KUKA KRL program: end_weld_respot.src

&ACCESS RVO3
&REL 155
&COMMENT end_weld_RESPOT
&PARAM DISKPATH = KRC:\R1\Program\SubRotinas
DEF end_weld_RESPOT( )
;
; FIM DO PROCESSO DE SOLDAGEM
;FOLD PULSE 3333 'R5 trabalho concluido' State=TRUE Time=3 sec;%{PE}%R 8.2.20,%MKUKATPBASIS,%COUT,%VPULSE,%P 2:3333, 3:R5 trabalho concluido, 5:TRUE, 6:, 8:3
PULSE($OUT[3333], TRUE,3)
;ENDFOLD
;
;FOLD WAIT Time=2 sec;%{PE}%R 8.2.20,%MKUKATPBASIS,%CWAIT,%VWAIT,%P 3:2
WAIT SEC 2
;ENDFOLD

END
